(* Copyright 2017 Cimpress

Licensed under the Apache License, Version 2.0 (the "License");
you may not use this file except in compliance with the License.
You may obtain a copy of the License at

http://www.apache.org/licenses/LICENSE-2.0

Unless required by applicable law or agreed to in writing, software
distributed under the License is distributed on an "AS IS" BASIS,
WITHOUT WARRANTIES OR CONDITIONS OF ANY KIND, either express or implied.
See the License for the specific language governing permissions and
limitations under the License. *)

TYPE T_Bl_LibHandleRow :
STRUCT
	pQueueHandle :ARRAY[0..BasLog.cMAX_CLIENTS] OF POINTER TO T_Queue_Info; // handle for access buffer
	usiRequest: USINT; // information if task allready requested a handle
END_STRUCT
END_TYPE

(* stored: Version 1.1.0.1, ProductVersion 3.1.4019.2
   DUT T_Bl_LibHandleRow: Id {a44ad8a8-5f74-495d-b7de-f0e7293b572f} *)
